FUNCTION_BLOCK fbHSV
VAR_INPUT
	Interlock_1 : BOOL;
	Interlock_2 : BOOL;
	Interlock_3 : BOOL;
	Interlock_4 : BOOL;
	Interlock_5 : BOOL;
	Interlock_6 : BOOL;
	Interlock_7 : BOOL;

	AutoCmd : BOOL;
END_VAR
VAR_OUTPUT
	AutoMan : BOOL;
	FB_Open : BOOL;
	FB_Travelling : BOOL;
	FB_Close : BOOL;
	Alarm : BOOL;
	Alarm_ID : INT;
END_VAR
VAR
	CmdOut AT %Q* : BOOL;
	OpenSenIn AT %I*: BOOL;
	CloseSenIn AT %I* : BOOL;
	Interlock_OK : BOOL;
	AutoReq : BOOL;
	ManReq : BOOL;
	ManOpenReq : BOOL;
	ManCloseReq : BOOL;
	ManCmd : BOOL;
	strInterlock_1 : STRING;
	strInterlock_2 : STRING;
	strInterlock_3 : STRING;
	strInterlock_4 : STRING;
	strInterlock_5 : STRING;
	strInterlock_6 : STRING;
	strInterlock_7 : STRING;
	strAutoMan : STRING;
	strOpenTravClose : STRING;
	idxOpenTravClose : INT;
	EnableAlarm : BOOL;
	AlarmDelayTime : TIME := T#5S;
	tonAlarmDelay : TON;
	
	SimHSV : fbSimHSV;
END_VAR
VAR // added by the converter: edge detectors and wires of the graphical bodies
    _w1, _w2, _w3 : BOOL;
END_VAR

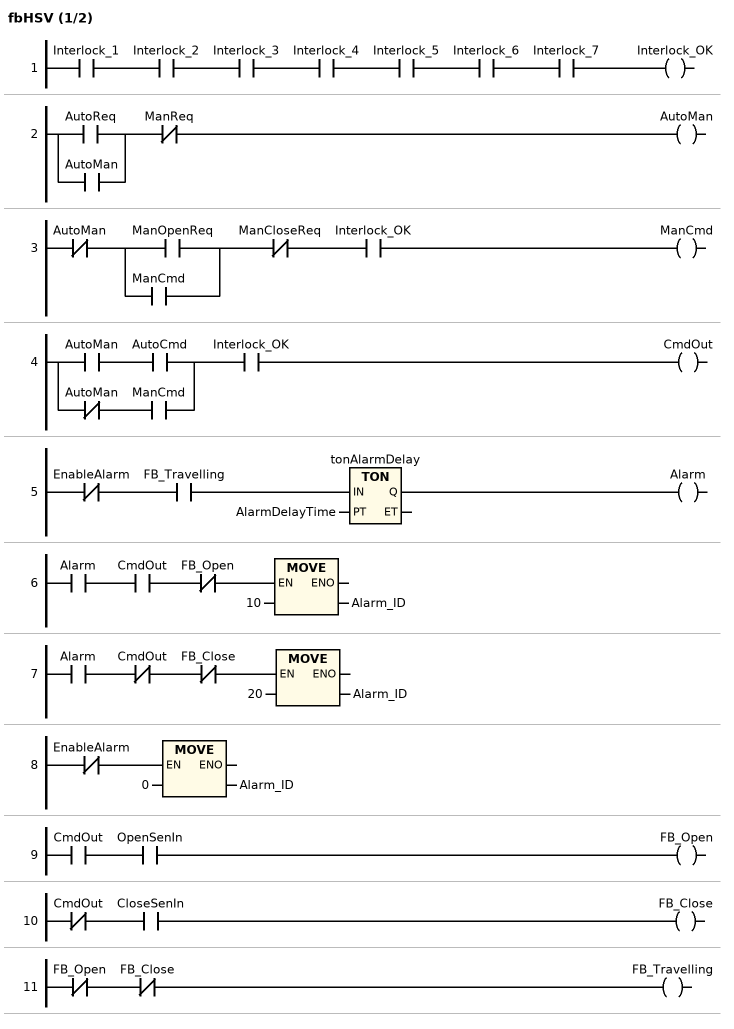
// NETWORK 1
Interlock_OK := Interlock_1 AND Interlock_2 AND Interlock_3 AND Interlock_4 AND Interlock_5 AND Interlock_6 AND Interlock_7;

// NETWORK 2
AutoMan := (AutoReq OR AutoMan) AND NOT ManReq;

// NETWORK 3
ManCmd := NOT AutoMan AND (ManOpenReq OR ManCmd) AND NOT ManCloseReq AND Interlock_OK;

// NETWORK 4
CmdOut := (AutoMan AND AutoCmd OR NOT AutoMan AND ManCmd) AND Interlock_OK;

// NETWORK 5
tonAlarmDelay(IN := NOT EnableAlarm AND FB_Travelling, PT := AlarmDelayTime); // TON
Alarm := tonAlarmDelay.Q;

// NETWORK 6
IF Alarm AND CmdOut AND NOT FB_Open THEN Alarm_ID := 10; END_IF

// NETWORK 7
IF Alarm AND NOT CmdOut AND NOT FB_Close THEN Alarm_ID := 20; END_IF

// NETWORK 8
IF NOT EnableAlarm THEN Alarm_ID := 0; END_IF

// NETWORK 9
FB_Open := CmdOut AND OpenSenIn;

// NETWORK 10
FB_Close := NOT CmdOut AND CloseSenIn;

// NETWORK 11
FB_Travelling := NOT FB_Open AND NOT FB_Close;

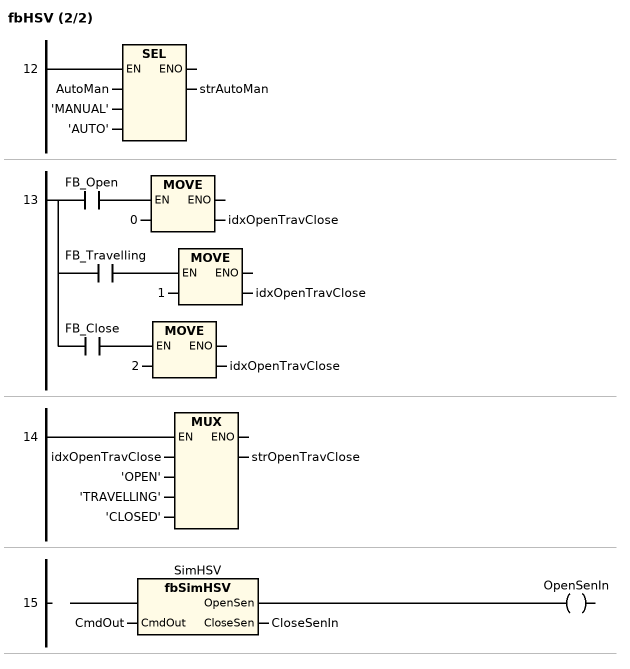
// NETWORK 12
strAutoMan := SEL(AutoMan, 'MANUAL', 'AUTO');

// NETWORK 13
_w1 := FB_Open;
IF _w1 THEN idxOpenTravClose := 0; END_IF
_w2 := FB_Travelling;
IF _w2 THEN idxOpenTravClose := 1; END_IF
_w3 := FB_Close;
IF _w3 THEN idxOpenTravClose := 2; END_IF
(* _w1 OR _w2 OR _w3; result not used *)

// NETWORK 14
strOpenTravClose := MUX(idxOpenTravClose, 'OPEN', 'TRAVELLING', 'CLOSED');

// NETWORK 15
SimHSV(CmdOut := CmdOut, CloseSen => CloseSenIn); // fbSimHSV
OpenSenIn := SimHSV.OpenSen;

END_FUNCTION_BLOCK

(* stored: Version 1.1.0.1, ProductVersion 3.1.4022.17
   POU fbHSV: Id {83158110-a4a6-4d8f-9eec-f01cc076b406}, SpecialFunc None *)
